// TIA Portal V16 export
// export: Created 2024-09-05T17:39:25.0930069Z, ExportSetting WithDefaults, DisplayName Totally Integrated Automation Portal, DisplayVersion V16 Update 6, DisplayName TIA Portal Version Control Interface, DisplayVersion V16 Update 2, DisplayName TIA Portal Openness, DisplayVersion V16 Update 6, DisplayName STEP 7 Professional, DisplayVersion V16 Update 6, DisplayName STEP 7 Safety, DisplayVersion V16, DisplayName WinCC Advanced, DisplayVersion V16 Update 6
DATA_BLOCK "MII_Interface_Data"   // DB2022
{ S7_Optimized_Access := 'TRUE' }
VERSION : 0.1
// stored: AutoNumber false, DBAccessibleFromOPCUA true, IsOnlyStoredInLoadMemory false, IsRetainMemResEnabled false, IsWriteProtectedInAS false, MemoryReserve 100
   VAR
      MII_METHODS { ExternalAccessible := 'False'; ExternalVisible := 'False'; ExternalWritable := 'False'} : Struct
         MethodStatusList { ExternalAccessible := 'False'; ExternalVisible := 'False'; ExternalWritable := 'False'} : Array[0..9] of DWord;
         MethodResultList { ExternalAccessible := 'False'; ExternalVisible := 'False'; ExternalWritable := 'False'} : Array[0..9] of DWord;
         M000_PRODUCTION_DECLARATION { ExternalAccessible := 'False'; ExternalVisible := 'False'; ExternalWritable := 'False'} : Struct
            Inputs { ExternalAccessible := 'False'; ExternalVisible := 'False'; ExternalWritable := 'False'; S7_SetPoint := 'True'} : "MII_Interface.MII_METHODS.M000_PRODUCTION_DECLARATION.Inputs";   // the definition of the input argument of method 1:Destinations.1:PRODUCTION_DECLARATION
            Outputs { ExternalAccessible := 'False'; ExternalVisible := 'False'; ExternalWritable := 'False'; S7_SetPoint := 'True'} : "MII_Interface.MII_METHODS.M000_PRODUCTION_DECLARATION.Outputs";   // the definition of the output arguments of method 1:Destinations.1:PRODUCTION_DECLARATION
         END_STRUCT;
         M001_GET_LOCAL_TIME { ExternalAccessible := 'False'; ExternalVisible := 'False'; ExternalWritable := 'False'} : Struct
            Outputs { ExternalAccessible := 'False'; ExternalVisible := 'False'; ExternalWritable := 'False'; S7_SetPoint := 'True'} : "MII_Interface.MII_METHODS.M001_GET_LOCAL_TIME.Outputs";   // the definition of the output arguments of method 2:Destinations.2:2_GET_LOCAL_TIME
         END_STRUCT;
         M101_SCRAP_DECLARATION { ExternalAccessible := 'False'; ExternalVisible := 'False'; ExternalWritable := 'False'} : Struct
            Inputs { ExternalAccessible := 'False'; ExternalVisible := 'False'; ExternalWritable := 'False'; S7_SetPoint := 'True'} : "MII_Interface.MII_METHODS.M101_SCRAP_DECLARATION.Inputs";   // the definition of the input argument of method 2:Destinations.2:1_SCRAP_DECLARATION
            Outputs { ExternalAccessible := 'False'; ExternalVisible := 'False'; ExternalWritable := 'False'; S7_SetPoint := 'True'} : "MII_Interface.MII_METHODS.M101_SCRAP_DECLARATION.Outputs";   // the definition of the output arguments of method 2:Destinations.2:1_SCRAP_DECLARATION
         END_STRUCT;
         M003_GENERATE_ALERT { ExternalAccessible := 'False'; ExternalVisible := 'False'; ExternalWritable := 'False'} : Struct
            Inputs { ExternalAccessible := 'False'; ExternalVisible := 'False'; ExternalWritable := 'False'; S7_SetPoint := 'True'} : "MII_Interface.MII_METHODS.M003_GENERATE_ALERT.Inputs";   // the definition of the input argument of method 2:Destinations.2:3_GENERATE_ALERT
            Outputs { ExternalAccessible := 'False'; ExternalVisible := 'False'; ExternalWritable := 'False'; S7_SetPoint := 'True'} : "MII_Interface.MII_METHODS.M003_GENERATE_ALERT.Outputs";   // the definition of the output arguments of method 2:Destinations.2:3_GENERATE_ALERT
         END_STRUCT;
         M102_REWORK_DECLARATION { ExternalAccessible := 'False'; ExternalVisible := 'False'; ExternalWritable := 'False'} : Struct
            Inputs { ExternalAccessible := 'False'; ExternalVisible := 'False'; ExternalWritable := 'False'; S7_SetPoint := 'True'} : "MII_Interface.MII_METHODS.M102_REWORK_DECLARATION.Inputs";   // the definition of the input argument of method 2:Destinations.2:4_REWORK_DECLARATION
            Outputs { ExternalAccessible := 'False'; ExternalVisible := 'False'; ExternalWritable := 'False'; S7_SetPoint := 'True'} : "MII_Interface.MII_METHODS.M102_REWORK_DECLARATION.Outputs";   // the definition of the output arguments of method 2:Destinations.2:4_REWORK_DECLARATION
         END_STRUCT;
         M002_GET_PLANTS { ExternalAccessible := 'False'; ExternalVisible := 'False'; ExternalWritable := 'False'} : Struct
            Outputs { ExternalAccessible := 'False'; ExternalVisible := 'False'; ExternalWritable := 'False'; S7_SetPoint := 'True'} : "MII_Interface.MII_METHODS.M002_GET_PLANTS.Outputs";   // the definition of the output arguments of method 2:Destinations.2:M005_GET_PLANTS
         END_STRUCT;
         M004_NTRS { ExternalAccessible := 'False'; ExternalVisible := 'False'; ExternalWritable := 'False'} : Struct
            Inputs { ExternalAccessible := 'False'; ExternalVisible := 'False'; ExternalWritable := 'False'; S7_SetPoint := 'True'} : "MII_Interface.MII_METHODS.M004_NTRS.Inputs";   // the definition of the input argument of method 2:Destinations.2:M006_NTRS
            Outputs { ExternalAccessible := 'False'; ExternalVisible := 'False'; ExternalWritable := 'False'; S7_SetPoint := 'True'} : "MII_Interface.MII_METHODS.M004_NTRS.Outputs";   // the definition of the output arguments of method 2:Destinations.2:M006_NTRS
         END_STRUCT;
         M103_PY { ExternalAccessible := 'False'; ExternalVisible := 'False'; ExternalWritable := 'False'} : Struct
            Inputs { ExternalAccessible := 'False'; ExternalVisible := 'False'; ExternalWritable := 'False'; S7_SetPoint := 'True'} : "MII_Interface.MII_METHODS.M103_PY.Inputs";   // the definition of the input argument of method 2:Destinations.2:M103_PY
            Outputs { ExternalAccessible := 'False'; ExternalVisible := 'False'; ExternalWritable := 'False'; S7_SetPoint := 'True'} : "MII_Interface.MII_METHODS.M103_PY.Outputs";   // the definition of the output arguments of method 2:Destinations.2:M103_PY
         END_STRUCT;
         M005_VARIABILITY { ExternalAccessible := 'False'; ExternalVisible := 'False'; ExternalWritable := 'False'} : Struct
            Inputs { ExternalAccessible := 'False'; ExternalVisible := 'False'; ExternalWritable := 'False'; S7_SetPoint := 'True'} : "MII_Interface.MII_METHODS.M005_VARIABILITY.Inputs";   // the definition of the input argument of method 2:Destinations.2:M005_VARIABILITY
            Outputs { ExternalAccessible := 'False'; ExternalVisible := 'False'; ExternalWritable := 'False'; S7_SetPoint := 'True'} : "MII_Interface.MII_METHODS.M005_VARIABILITY.Outputs";   // the definition of the output arguments of method 2:Destinations.2:M005_VARIABILITY
         END_STRUCT;
         M006_MII_GET_PART_HMAC { ExternalAccessible := 'False'; ExternalVisible := 'False'; ExternalWritable := 'False'} : Struct
            Inputs { ExternalAccessible := 'False'; ExternalVisible := 'False'; ExternalWritable := 'False'; S7_SetPoint := 'True'} : "MII_Interface.MII_METHODS.M006_MII_GET_PART_HMAC.Inputs";   // the definition of the input argument of method 2:Destinations.2:M006_MII_GET_PART_HMAC
            Outputs { ExternalAccessible := 'False'; ExternalVisible := 'False'; ExternalWritable := 'False'; S7_SetPoint := 'True'} : "MII_Interface.MII_METHODS.M006_MII_GET_PART_HMAC.Outputs";   // the definition of the output arguments of method 2:Destinations.2:M006_MII_GET_PART_HMAC
         END_STRUCT;
      END_STRUCT;
   END_VAR
BEGIN
END_DATA_BLOCK
